FUNCTION_BLOCK ASRT_SRT_TO_3EVENTS (* Composite FB for convert ASRT to 3 EVENTS *)
  (* Standard: 61499-2; Description: Copyright (c) 2026 HR Agrartechnik GmbH This program and the accompanying materials are made available under the terms of the Eclipse Public License 2.0 which is available at https://www.eclipse.org/legal/epl-2.0/ SPDX-License-Identifier: EPL-2.0 *)
  (* Version 1.0, 2026-09-03, Franz Höpfinger, HR Agrartechnik GmbH *)
  PACKAGE adapter::conversion::unidirectional;
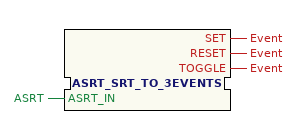
  EVENT_OUTPUT
    SET; (* Set / Switch on *)
    RESET; (* Reset / Switch off *)
    TOGGLE; (* Toggle / Switch output *)
  END_EVENT
  SOCKETS
    ASRT_IN : adapter::types::unidirectional::ASRT; (* Adapter Input *)
  END_SOCKETS
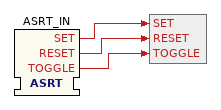
  EVENT_CONNECTIONS
    ASRT_IN.SET TO SET;
    ASRT_IN.RESET TO RESET;
    ASRT_IN.TOGGLE TO TOGGLE;
  END_CONNECTIONS
END_FUNCTION_BLOCK
